% RSLogix 500 project PROBLOM 4 LAB 1 AUTO_BAK000.RSS, saved by version 8.30.00.16 %
PROJECT "UNTITLED"    % processor: Bul.1763 MicroLogix 1100 Series B %

PROGRAM FILES
  LAD 2   8 rungs

DATA FILES
  O0 OUTPUT  4 elements
  I1 INPUT  6 elements
  S2 STATUS  66 elements
  B3 BINARY  1 elements
  T4 TIMER  1 elements
  C5 COUNTER  1 elements
  R6 CONTROL  1 elements
  N7 INTEGER  1 elements
  F8 FLOAT  1 elements

LADDER 2
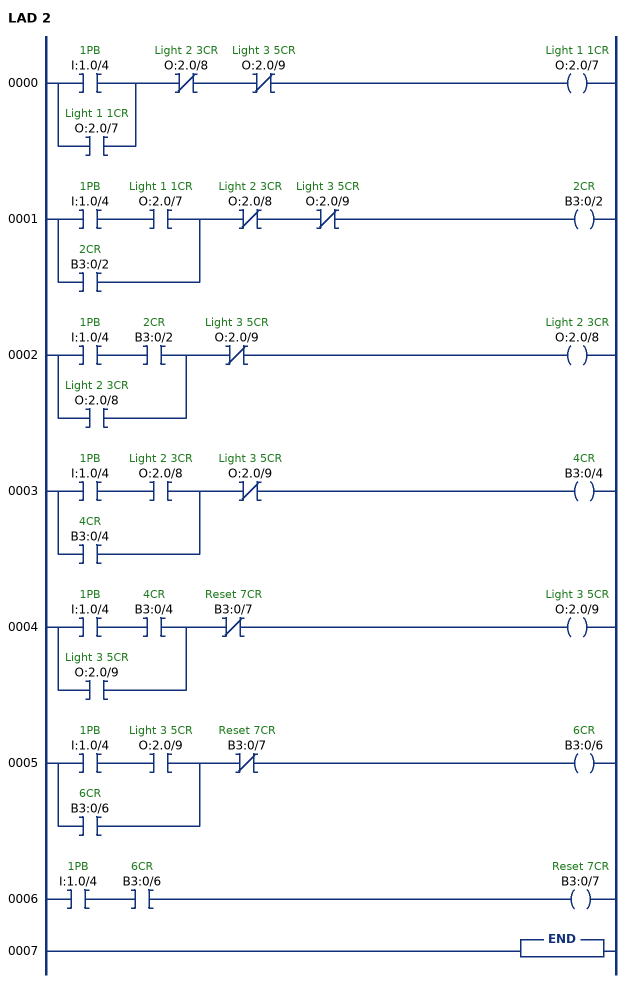
% Rung: 0 %  % edit flag set %
SOR BST XIC I:1.0/4 NXB XIC O:2.0/7 BND XIO O:2.0/8 XIO O:2.0/9 OTE O:2.0/7 EOR
%   I:1.0/4  1PB %
%   O:2.0/7  1CR  "Light 1" %
%   O:2.0/8  3CR  "Light 2" %
%   O:2.0/9  5CR  "Light 3" %
% Rung: 1 %  % edit flag set %
SOR BST XIC I:1.0/4 XIC O:2.0/7 NXB XIC B3:0/2 BND XIO O:2.0/8 XIO O:2.0/9 OTE B3:0/2 EOR
%   I:1.0/4  1PB %
%   O:2.0/7  1CR  "Light 1" %
%   B3:0/2  2CR %
%   O:2.0/8  3CR  "Light 2" %
%   O:2.0/9  5CR  "Light 3" %
% Rung: 2 %  % edit flag set %
SOR BST XIC I:1.0/4 XIC B3:0/2 NXB XIC O:2.0/8 BND XIO O:2.0/9 OTE O:2.0/8 EOR
%   I:1.0/4  1PB %
%   B3:0/2  2CR %
%   O:2.0/8  3CR  "Light 2" %
%   O:2.0/9  5CR  "Light 3" %
% Rung: 3 %  % edit flag set %
SOR BST XIC I:1.0/4 XIC O:2.0/8 NXB XIC B3:0/4 BND XIO O:2.0/9 OTE B3:0/4 EOR
%   I:1.0/4  1PB %
%   O:2.0/8  3CR  "Light 2" %
%   B3:0/4  4CR %
%   O:2.0/9  5CR  "Light 3" %
% Rung: 4 %  % edit flag set %
SOR BST XIC I:1.0/4 XIC B3:0/4 NXB XIC O:2.0/9 BND XIO B3:0/7 OTE O:2.0/9 EOR
%   I:1.0/4  1PB %
%   B3:0/4  4CR %
%   O:2.0/9  5CR  "Light 3" %
%   B3:0/7  7CR  "Reset" %
% Rung: 5 %  % edit flag set %
SOR BST XIC I:1.0/4 XIC O:2.0/9 NXB XIC B3:0/6 BND XIO B3:0/7 OTE B3:0/6 EOR
%   I:1.0/4  1PB %
%   O:2.0/9  5CR  "Light 3" %
%   B3:0/6  6CR %
%   B3:0/7  7CR  "Reset" %
% Rung: 6 %  % edit flag set %
SOR XIC I:1.0/4 XIC B3:0/6 OTE B3:0/7 EOR
%   I:1.0/4  1PB %
%   B3:0/6  6CR %
%   B3:0/7  7CR  "Reset" %
% Rung: 7 %
SOR END EOR
